FUNCTION_BLOCK "fbAdd"
{ S7_Optimized_Access := 'TRUE' }
VERSION : 0.1
   VAR_INPUT
      "Input 1" : Real;
      "Input 2" : Real;
   END_VAR

   VAR_OUTPUT
      Sum : Real;
   END_VAR


BEGIN
	#Sum := #"Input 1" + #"Input 2";
END_FUNCTION_BLOCK

